Staubli VAL3: CartesianTrajPtMsg.pjx

--- CartesianTrajPtMsg.pjx ---
Parameters version=s7.7.2 stackSize=5000 millimeterUnit=true
Program file=start.pgx
Program file=stop.pgx
Data file=CartesianTrajPtMsg.dtx
Type name=Body path=Disk://ros_libs/Body/Body.pjx
Type name=Header path=Disk://ros_libs/Header/Header.pjx
Type name=Prefix path=Disk://ros_libs/Prefix/Prefix.pjx
Type name=CartesianTrajPt path=Disk://ros_libs/CartesianTrajPt/CartesianTrajPt.pjx

--- CartesianTrajPtMsg.dtx ---
public Header header
  [0]
    num nMsgType
    num nCommType
    num nReplyCode
    num nData[12]
public CartesianTrajPt cartesianTrajPt
  [0]
    num nSeq
    num nPosition[3]
    num nOrientation[4]
    num nVelocity
    num nAcceleration
    num nBlendingRadius
    num nDuration
public Prefix prefix
  [0]
    num nLength
    num nData[4]
public Body body
  [0]
    num nData[64]
